// TwinCAT 3 PLC project Test
// ProgramVersion: 3.1.4024.0
// libraries:
//   Festo_HomingLibrary, * (Festo)
//   Tc2_EtherCAT, * (Beckhoff Automation GmbH)
//   Tc2_MC2, * (Beckhoff Automation GmbH)
//   Tc2_Standard, * (Beckhoff Automation GmbH)
//   Tc2_System, * (Beckhoff Automation GmbH)
//   Tc3_Module, * (Beckhoff Automation GmbH)
// project tree:
//   / PlcTask.TcTTO
//   POUs/ CMMT_AS_EtherCAT.TcPOU, MAIN.TcPOU
// real-time tasks:
//   TASK PlcTask: cycle T#10ms, priority 20, ADS port 350
// motion (NC):
//   TASK NC-Task 1 SAF: cycle T#2ms, priority 4, ADS port 501
//   TASK NC-Task 1 SVB: cycle T#10ms, priority 9, ADS port 511
//   AXIS Axis 1 (id 1)
//     OtherSettings: AllowMotionCmdToSlave=true
//     encoder EncType=19
//       EncPara: ScaleFactorNumerator=1e-06, MaxCount=#xffffffff
//     drive DrvType=16
//       DrvPara: MaxCount=#xffffffff, DriveControlDWord=#x00000100
//         Analog: TorqueSetpointScale=10, ScaleFactorActTorque=0.1
//         TimeComp: TaskDelayCycles=1
//     controller CtrType=1
//       CtrPara: PriorControlFactor=1
//         Observer: BandWidth=20
//   AXIS Axis 2 (id 2)
//     OtherSettings: AllowMotionCmdToSlave=true
//     encoder EncType=19
//       EncPara: ScaleFactorNumerator=1e-06, MaxCount=#xffffffff
//     drive DrvType=16
//       DrvPara: MaxCount=#xffffffff, DriveControlDWord=#x00000100
//         Analog: TorqueSetpointScale=10, ScaleFactorActTorque=0.1
//         TimeComp: TaskDelayCycles=1
//     controller CtrType=1
//       CtrPara: PriorControlFactor=1
//         Observer: BandWidth=20
//   AXIS Axis 3 (id 3)
//     OtherSettings: AllowMotionCmdToSlave=true
//     encoder EncType=19
//       EncPara: ScaleFactorNumerator=1e-05, MaxCount=#xffffffff
//     drive DrvType=16
//       DrvPara: MaxCount=#xffffffff, DriveControlDWord=#x00000100
//         Analog: TorqueSetpointScale=10, ScaleFactorActTorque=0.1
//         TimeComp: TaskDelayCycles=1
//     controller CtrType=1
//       CtrPara: PriorControlFactor=1
//         Observer: BandWidth=20
// I/O:
//   DEVICE Device 1 (EtherCAT), AmsNetId 5.50.156.206.2.1
//     Term 1 (EK1200) [EK1200-5000 EtherCAT Power supply (2A E-Bus)]
//       Term 3 (EK1110) [EK1110 EtherCAT extension]
//     Drive 1 (CMMT-AS) [CMMT-AS]
//     Drive 2 (CMMT-ST) [CMMT-ST]
//     Drive 3 (EMCA CiA402) [EMCA CiA402]

CONFIGURATION Test
    RESOURCE PLC ON TwinCAT3
        TASK PlcTask(INTERVAL := T#10ms, PRIORITY := 20);
        PROGRAM MAIN WITH PlcTask : MAIN;
    END_RESOURCE
END_CONFIGURATION

// ---- POUs/MAIN.TcPOU
PROGRAM MAIN
VAR
	CMMT_AS_EtherCAT	: CMMT_AS_EtherCAT;
	
END_VAR

CMMT_AS_EtherCAT();

END_PROGRAM

// ---- POUs/CMMT_AS_EtherCAT.TcPOU
FUNCTION_BLOCK CMMT_AS_EtherCAT
VAR
	MC_Power				: MC_Power;							// enable axis
	MC_Reset				: MC_Reset;							// reset axis if error is active
	Festo_MC_ReadAxisErr	: Festo_MC_ReadAxisError;			// read axis error
	Festo_MC_Home			: Festo_MC_Home;					// start homing procedure 			
	MC_MovRel				: MC_MoveRelative;					// move relative
	
	Axis					: AXIS_REF;							// axis reference structure	
	Start					: BOOL;								// start statemachine
	ReadAxisError			: BOOL;								// start reading axis error
	Step					: UINT;								// statemachine
	Counter					: DINT;								// counter how many times statemachine was finished successfully
END_VAR

(*cyclic call of function blocks*)
MC_Power(Axis:= Axis);
MC_Reset(Axis:= Axis);
Festo_MC_Home(Axis:= Axis);
Festo_MC_ReadAxisErr(Axis:= Axis, Enable:=ReadAxisError);
MC_MovRel(Axis:= Axis, Distance:= 25, Velocity:= 15, Acceleration:= 100, Deceleration:= 100, Jerk:= 300);

// reset statemachine if start is FALSE
IF NOT START THEN
	Step	:= 0;
END_IF

(*Statemachine*)
CASE Step OF
	0: // init
		MC_Power.Enable				:= FALSE;
		MC_Reset.Execute			:= FALSE;
		Festo_MC_Home.Execute		:= FALSE;
		MC_MovRel.Execute			:= FALSE;
		
		IF Start THEN
			Step					:= 1;
		END_IF
	
	1: // enable
		MC_Power.Enable				:= TRUE;
		MC_Power.Enable_Positive	:= TRUE;
		MC_Power.Enable_Negative	:= TRUE;

		IF MC_Power.Status THEN
			Step					:= 20;
		ELSIF MC_Power.Error THEN
			Step					:= 10;	
		END_IF
		
	10: // reset
		MC_Reset.Execute			:= TRUE;
		
		IF MC_Reset.Done THEN
			MC_Reset.Execute		:= FALSE;
			Step					:= 0;
		END_IF
	
	20: // start homing
		Festo_MC_Home.Execute				:= TRUE;

		IF Festo_MC_Home.Done AND Axis.NcToPlc.ActPos > -1.5 AND Axis.NcToPlc.ActPos < 1.5 THEN
			Festo_MC_Home.Execute	:= FALSE;	
			Step					:= 30;
		END_IF

	30: // move rel no. 1
		MC_MovRel.Execute			:= TRUE;
		
		IF MC_MovRel.Done THEN
			MC_MovRel.Execute		:= FALSE;
			Step					:= 40;
		END_IF
		
	40: // move rel no. 2	
		MC_MovRel.Execute			:= TRUE;
		
		IF MC_MovRel.Done THEN
			MC_MovRel.Execute		:= FALSE;
			Counter					:= Counter + 1;
			Step					:= 20;
		END_IF	
END_CASE

END_FUNCTION_BLOCK
